TYPE "Inverter_controller"
VERSION : 0.1
   STRUCT
      Enabled : Bool;   // Operator/HMI enable - manual, never overwritten by automatic logic
      RemReady : Bool;
      Error : Bool;
      CommError : Bool;
      Available : Bool;   // Combined online criteria, written ONCE by FC_PPC_InverterMonitor (step 1):
                           // Enabled AND RemReady AND NOT Error AND NOT CommError AND PwrOffReas=0 AND ELECTRIC_OK.
                           // PowerDistribution / ReactiveControl read this instead of re-deriving the criteria.
      OperMode : DInt;   // Operating state of the inverter, setpoint
      Wactive : DInt;
      Qactive : DInt;
      WMode : DInt;   // Selection of procedure for setpoint for active power
      VArMode : DInt;   // Selection of procedure for setpoint for reactive power
      WSpt : DInt;   // Inverter active power setpoint.
      VArSpt : DInt;   // Inverter reactive power setpoint (if Q control).
      PFSpt : DInt;   // Inverter power factor setpoint (if PF control).
      WAval : DInt;   // Available active power.
      VArAval : DInt;   // Available reactive power.
      PwrOffReas : DInt;   // Detect why inverter disconnected.
      DrtStt : DInt;   // Derating state.
      ErrClr : DInt;
      WSptMax : Real;   // Plant P ceiling from grid operator (kW) - maps to UID2 addr 4039
      WSptMin : Real;   // Plant P floor kW - negative valid for load/charge mode - maps to UID2 addr 4041
   END_STRUCT;

END_TYPE

